FUNCTION_BLOCK L2_OPBuffer (* Basic Function Block Type *)
  (* Standard: 61499-2 *)
  (* Version 0.0, 2014-11-28, EQUEROL, UJI *)
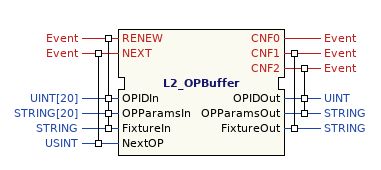
  EVENT_INPUT
    RENEW WITH OPIDIn, OPParamsIn, FixtureIn; (* Initialization Request *)
    NEXT WITH NextOP; (* Normal Execution Request *)
  END_EVENT
  EVENT_OUTPUT
    CNF0; (* Renew confirmation *)
    CNF1 WITH FixtureOut; (* Initialization Confirm *)
    CNF2 WITH OPIDOut, OPParamsOut; (* Execution Confirmation *)
  END_EVENT
  VAR_INPUT
    OPIDIn : ARRAY [0..19] OF UINT := [0,0,0,0,0,0,0,0,0,0,0,0,0,0,0,0,0,0,0,0]; (* Operation identifiers *)
    OPParamsIn : ARRAY [0..19] OF STRING; (* Operation parameters *)
    FixtureIn : STRING; (* Setup fixture *)
    NextOP : USINT; (* Next operation position within the buffer *)
  END_VAR
  VAR_OUTPUT
    OPIDOut : UINT := 0; (* Operation to be executed identifier *)
    OPParamsOut : STRING; (* Operation to be executed parameters *)
    FixtureOut : STRING; (* Fixture to be used in this setup *)
  END_VAR
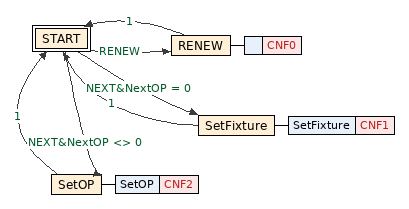
  EC_STATES
    START; (* Initial State *)
    RENEW : -> CNF0; (* Normal execution *)
    SetFixture : SetFixture -> CNF1;
    SetOP : SetOP -> CNF2;
  END_STATES
  EC_TRANSITIONS
    START TO RENEW := RENEW;
    RENEW TO START := 1;
    START TO SetFixture := NEXT&NextOP = 0;
    START TO SetOP := NEXT&NextOP <> 0;
    SetOP TO START := 1;
    SetFixture TO START := 1;
  END_TRANSITIONS
  ALGORITHM SetFixture IN ST: (* new algorithm *)
FixtureOut := FixtureIn;
  END_ALGORITHM
  ALGORITHM SetOP IN ST: (* new algorithm *)
OPIDOut := OPIDIn[NextOP -1];
OPParamsOut := OPParamsIn[NextOP - 1];
  END_ALGORITHM
END_FUNCTION_BLOCK
